   VAR
      b_HmiCmdModAut { ExternalVisible := 'False'} : Bool;   //  command change mode to AUTO
      b_HmiCmdModMan { ExternalVisible := 'False'} : Bool;   //  command change mode to MANUAL
      b_HmiCmdModDis { ExternalVisible := 'False'} : Bool;   //  command change mode to DISABLED
      b_HmiCmdSim { ExternalVisible := 'False'} : Bool;   //  toggle simulation mode
      b_HmiCmdRst { ExternalVisible := 'False'} : Bool;   //  reset alarms
      b_HmiCmdAutoSim { ExternalVisible := 'False'} : Bool;   //  toggle automatic simulation value
      b_HmiCmdFwd { ExternalVisible := 'False'} : Bool;   //  command start forward
      b_HmiCmdRev { ExternalVisible := 'False'} : Bool;   //  command start reversed
      b_HmiCmdStp { ExternalVisible := 'False'} : Bool;   //  command stop
      b_HmiCmdRstActOpe { ExternalVisible := 'False'} : Bool;   //  reset actuation counter and operating hours
      b_StaModAut { ExternalVisible := 'False'} : Bool;   //  state AUTOMATIC
      b_StaModMan { ExternalVisible := 'False'} : Bool := TRUE;   //  state MANUAL
      b_StaModDis { ExternalVisible := 'False'} : Bool;   //  state DISABLED
      b_StaSim { ExternalVisible := 'False'} : Bool;   //  state simulation ON
      b_StaIlOn { ExternalVisible := 'False'} : Bool;   //  state interlock ON : 1 = interlocked (prevents forward)
      b_StaIlRev : Bool;   //  state interlock ON : 1 = interlocked (prevents reverse)
      b_StaSaf { ExternalVisible := 'False'} : Bool;   //  state safety : 1 = error (valve to safety position)
      b_StaAutoSim { ExternalVisible := 'False'} : Bool;   //  Auto sim (Ir_ActSpd simulated)
      b_ReqFwd { ExternalVisible := 'False'} : Bool;   //  output forward
      b_ReqRev { ExternalVisible := 'False'} : Bool;   //  output reversed
      b_StaSpdOk { ExternalVisible := 'False'} : Bool;   //  speed (setpoint) reached
      b_StaAlm { ExternalVisible := 'False'} : Bool;   //  general alarm
      b_StaWrn { ExternalVisible := 'False'} : Bool;   //  general warning
      b_CfgAnaSpdPres { ExternalVisible := 'False'} : Bool;   //  configuration : analog speed feedback present
      b_CfgEnRev { ExternalVisible := 'False'} : Bool;   //  configuration : reversed direction enabled
      b_CfgHldMod { ExternalVisible := 'False'} : Bool;   //  Configuration : status bit mode after reset (1 = auto, 0 = manual)
      b_CfgPushToRun { ExternalVisible := 'False'} : Bool;
      b_CfgDisableSim { ExternalVisible := 'False'} : Bool;
      b_CfgStopArea { ExternalVisible := 'False'} : Bool;
      b_AlmToFb { ExternalVisible := 'False'} : Bool;   //  alarm time out feedback
      b_AlmToRun { ExternalVisible := 'False'} : Bool;   //  alarm run time too long
      b_AlmIs { ExternalVisible := 'False'} : Bool;   //  alarm isolation switch
      b_AlmMps { ExternalVisible := 'False'} : Bool;   //  alarm motor protection switch
      b_AlmDevFlt { ExternalVisible := 'False'} : Bool;   //  alarm device fault
      b_ReqAut { ExternalVisible := 'False'} : Bool;   //  automatic mode requested
      b_ReqMan { ExternalVisible := 'False'} : Bool;   //  manual mode requested
      b_ReqDis { ExternalVisible := 'False'} : Bool;   //  disabled mode requested
      b_TFbSpd { ExternalVisible := 'False'} : Bool;   //  timer finished, feedback monitoring Pos1
      b_SpChange : Bool;
      r_SpSel { ExternalVisible := 'False'} : Real;   //  selected setpoint
      r_SpPrev : Real;
      r_DevMax { ExternalVisible := 'False'} : Real;
      r_DevMin { ExternalVisible := 'False'} : Real;
      b_CmdManFwd { ExternalVisible := 'False'} : Bool;   //  internal memo : manual command forward
      b_CmdManRev { ExternalVisible := 'False'} : Bool;   //  internal memo : manual command reversed
      b_CmdAutFwd { ExternalVisible := 'False'} : Bool;   //  internal memo : automatic command forward
      b_CmdAutRev { ExternalVisible := 'False'} : Bool;   //  internal memo : automatic command reversed
      b_CmdFwd { ExternalVisible := 'False'} : Bool;   //  internal memo : command forward (combined manual and auto)
      b_CmdRev { ExternalVisible := 'False'} : Bool;   //  internal memo : command reversed(combined manual and auto)
      b_FbErrSpd { ExternalVisible := 'False'} : Bool;   //  internal memo : error detection feedback analogue value
      b_TFbOnOut { ExternalVisible := 'False'} : Bool;   //  timer finished for feedback monitoring run (Fwd OR Rev)
      b_TFbOffOut { ExternalVisible := 'False'} : Bool;   //  timer finished for feedback monitoring stop
      b_TToRunOut { ExternalVisible := 'False'} : Bool;   //  timer finished for time out run
      i_TmrToRun : Int;   //  timer time out  run control
      i_TmrFbFwd { ExternalVisible := 'False'} : Int;   //  timer for feedback simulation (set) after start
      i_TmrFbRev { ExternalVisible := 'False'} : Int;   //  timer for feedback simulation (reset) after stop
      b_TFbFwdOut { ExternalVisible := 'False'} : Bool;   //  timer finished for simulation run (Fwd OR Rev)
      b_TFbRevOut { ExternalVisible := 'False'} : Bool;   //  timer finished for simulation stopped
      FB_UTIL_TON_Del_1 : "FB_UTIL_TON_Sec";
      FB_UTIL_TON_Del_2 : "FB_UTIL_TON_Sec";
      FB_UTIL_TON_Del_3 : "FB_UTIL_TON_Sec";
      FB_UTIL_TON_Del_4 : "FB_UTIL_TON_Sec";
      b_Old_ob_Fwd : Bool;
      b_Old_ob_Rev : Bool;
      FB_UTIL_Work_H_Rst { ExternalVisible := 'False'} : "FB_UTIL_Work_H";
      FB_UTIL_Work_H_Tot { ExternalVisible := 'False'} : "FB_UTIL_Work_H";
      b_FbSimFwd : Bool;
      b_FbSimRev : Bool;
      b_FbErrFwd : Bool;
      b_FbErrRev : Bool;
      i_TmrFbSpd : Int;
      b_DisAlmWrn : Bool;
      b_dummy : Bool;
      i_dummy : Int;
      b_StaAlmNew : Bool;
      b_NoAlm : Bool;
      i_AlmAck : Int;
      b_DisAlmWrn_1 : Bool;
      b_RstAlm : Bool;
      b_HmiCmdLoc : Bool;
      b_HmiCmdRem : Bool;
      i_ErrCod : Int;
      b_LocGenEnab : Bool;
      b_DrwTest : Bool;
      b_DrwInst : Bool;
      b_DrwNotIns : Bool;
      b_ErrorCFW : Bool;
      b_RemoteM : Bool;
      b_ManutLocal { ExternalVisible := 'False'} : Bool;   // command change mode to "Manut.Local"
      b_FbRem : Bool;
      b_PerRemMod : Bool;
      I_HmiSta : Word;
      i_Category : Int := 1;   // Device alarm category setting
      b_NoFeedback : Bool;
      b_EnDisPump : Bool;   // Enable/Disable HMI option
   END_VAR

   VAR_TEMP
      di_AUX : DInt;   //  auxiliary double word for calculation of state or alarm word to HMI
   END_VAR


BEGIN
	// =============================================================================================================================
	// Purpose: Reditech standard typical for controlling a frequency driven motor
	// -----------------------------------------------------------------------------------------------------------------------------
	// Date (dd MMM yyyy)   Developer                   Version Comments/Reason for change
	// ..................   .........                   ....... ..........................
	// 13 Dec 2018          Bram Verheyen               08.0    Full review
	// 30 Jan 2019          Matthias De Staelen         08.1    Outputs can be high in simulation mode
	// 13 Mar 2020          Willian Barroso             08.2    Full review
	// 01 Jul 2021          Ivan Galhardoni             08.3    Added NoFeedback function
	// 03 Jul 2021          Ivan Galhardoni             08.4    Added No communication fault alarm and erase manual setpoint when interlock is incoming
	// =============================================================================================================================

	//============================================================================================
	#b_CfgAnaSpdPres := #Iw_Cfg.%X0;      // Analog speed feedback present
	#b_CfgEnRev := #Iw_Cfg.%X1;           // Reverse direction enable
	#b_CfgHldMod := #Iw_Cfg.%X2;          // Mode after reset (1 => auto, 0 => manual)
	#b_NoFeedback := #Iw_Cfg.%X3;         // No feedback configured
	#b_CfgPushToRun := #Iw_Cfg.%X8;
	#b_CfgDisableSim := #Iw_Cfg.%X10;
	#b_CfgStopArea := #Iw_Cfg.%X11;

	//============================================================================================
	#b_DisAlmWrn := #Ib_DisAlmWrn OR #IO_AreaCmd.Alm.Dis OR #b_StaModDis OR #b_StaSim;

	//============================================================================================
	#b_StaSaf := (#Iby_Saf <> 0) AND NOT #b_DisAlmWrn;
	#b_StaIlOn := (#Iby_IlFwd <> 0);
	//#b_StaIlRev := (#Iby_IlRev <> 0);

	//============================================================================================
	IF #b_StaSim THEN
	    #i_ErrCod := 15;
	    #b_LocGenEnab := TRUE;
	    #b_FbRem := TRUE;
	ELSE
	    #i_ErrCod := #Ii_CurFault;
	    #b_LocGenEnab := #Ib_LocGenEnab;
	    #b_FbRem := #Ib_FbRem;
	END_IF;

	#b_DrwTest := #Ib_DrwTest;
	#b_DrwInst := #Ib_DrwInst;

	//============================================================================================
	#b_HmiCmdModAut := #IOdi_HmiCmd.%X0;
	#b_HmiCmdModMan := #IOdi_HmiCmd.%X1;
	#b_HmiCmdModDis := #IOdi_HmiCmd.%X2;
	#b_HmiCmdSim := #IOdi_HmiCmd.%X3;
	#b_HmiCmdFwd := #IOdi_HmiCmd.%X4;
	#b_HmiCmdRev := #IOdi_HmiCmd.%X5;
	#b_HmiCmdStp := #IOdi_HmiCmd.%X6;
	#b_HmiCmdAutoSim := #IOdi_HmiCmd.%X8;
	#b_HmiCmdRstActOpe := #IOdi_HmiCmd.%X9;
	#b_ManutLocal := #IOdi_HmiCmd.%X10;

	//============================================================================================

	IF #b_CfgPushToRun THEN
	    #IOdi_HmiCmd := DWORD_TO_DINT(DINT_TO_DWORD(#IOdi_HmiCmd) AND 48);
	ELSE
	    #IOdi_HmiCmd := 0;
	END_IF;


	//============================================================================================
	IF  #IO_AreaCmd.Mode.AreaMode THEN
	    #b_ReqAut := #IO_AreaCmd.Mode.Auto;
	    #b_ReqMan := #IO_AreaCmd.Mode.Man;
	    #b_ReqDis := #IO_AreaCmd.Mode.Dis;

	ELSE
	    IF #b_CfgHldMod THEN
	        #b_ReqAut := #b_HmiCmdModAut;
	        #b_ReqMan := #b_HmiCmdModMan;
	        #b_ReqDis := #b_HmiCmdModDis;

	    ELSE
	        #b_ReqAut := #b_HmiCmdModAut AND NOT #b_StaAlm AND NOT #b_StaSaf;
	        #b_ReqMan := #b_HmiCmdModMan OR ((#b_StaAlm OR #b_StaSaf) AND NOT #b_StaModDis);
	        #b_ReqDis := #b_HmiCmdModDis;
	    END_IF;
	END_IF;
	IF (#b_ReqAut AND NOT #b_ReqMan AND NOT #b_ReqDis) THEN
	    #b_StaModAut := true;
	    #b_StaModMan := false;
	    #b_StaModDis := false;
	END_IF;
	IF (#b_ReqMan AND NOT #b_ReqAut AND NOT #b_ReqDis) THEN
	    #b_StaModAut := false;
	    #b_StaModMan := true;
	    #b_StaModDis := false;
	END_IF;
	IF (#b_ReqDis AND NOT #b_ReqMan AND NOT #b_ReqAut) THEN
	    #b_StaModAut := false;
	    #b_StaModMan := false;
	    #b_StaModDis := true;
	END_IF;

	//============================================================================================
	IF #IO_AreaCmd.Sim.ForceOn OR (#b_HmiCmdSim AND NOT #b_StaSim AND NOT #IO_AreaCmd.Sim.ForceOn AND NOT #IO_AreaCmd.Sim.ForceOff) THEN
	    #b_StaSim := true;
	    #b_HmiCmdSim := false; // reset of command necessary, else simulation will always be reset immediately by following instructions
	END_IF;
	IF #IO_AreaCmd.Sim.ForceOff OR (#b_HmiCmdSim AND #b_StaSim AND NOT #IO_AreaCmd.Sim.ForceOn AND NOT #IO_AreaCmd.Sim.ForceOff) THEN
	    #b_StaSim := false;
	    #b_HmiCmdSim := false;
	END_IF;

	//============================================================================================
	IF (#b_ReqFwd AND NOT #b_FbSimFwd)
	    OR (#b_ReqRev AND NOT #b_FbSimRev)
	    OR #b_HmiCmdStp
	    OR (NOT #b_ReqFwd AND NOT #b_ReqRev)
	    OR #b_StaIlOn
	    OR #b_StaAlm THEN
	    #b_FbSimFwd := false;
	    #b_FbSimRev := false;
	END_IF;

	IF ((#i_TmrFbFwd <= 1) OR #Ii_ParTFb = 0) AND #b_ReqFwd THEN
	    #b_FbSimFwd := true;
	    #b_FbSimRev := false;
	END_IF;

	IF ((#i_TmrFbRev <= 1) OR #Ii_ParTFb = 0) AND #b_ReqRev THEN
	    #b_FbSimFwd := false;
	    #b_FbSimRev := true;
	END_IF;

	//============================================================================================
	#r_DevMax := #r_SpSel + #Ir_ParCtlDev;
	#r_DevMin := #r_SpSel - #Ir_ParCtlDev;
	IF #b_StaSim AND #Ib_Pls1S THEN
	    IF (#IOr_SimSpd <= #r_DevMin) THEN
	        #IOr_SimSpd := #IOr_SimSpd + #Ir_ParCtlDev;
	    END_IF;
	    IF (#IOr_SimSpd >= #r_DevMax) THEN
	        #IOr_SimSpd := #IOr_SimSpd - #Ir_ParCtlDev;
	    END_IF;
	END_IF;

	// ACM: select speed
	IF #b_StaSim THEN
	    #Or_StaSpd := #IOr_SimSpd;
	ELSE
	    #Or_StaSpd := #Ir_ActSpd;
	END_IF;

	//============================================================================================
	#Ob_StaFwd := (NOT #b_StaSim AND #Ib_FbFwd)
	OR (#b_StaSim AND #b_FbSimFwd)
	OR (#b_NoFeedback AND #r_SpSel > 0.00);

	#Ob_StaRev := (NOT #b_StaSim AND #Ib_FbRev)
	OR (#b_StaSim AND #b_FbSimRev);

	#Ob_StaOff := NOT #Ob_StaFwd AND NOT #Ob_StaRev;

	#b_StaSpdOk := (NOT #b_CfgAnaSpdPres)
	OR (#b_CfgAnaSpdPres AND (#Or_StaSpd > #r_DevMin) AND (#Or_StaSpd < #r_DevMax));
	#Ob_SpdOk := #b_StaSpdOk AND NOT #b_StaAlm;

	//============================================================================================
	#b_SpChange := (#r_SpSel <> #r_SpPrev);
	#r_SpPrev := #r_SpSel;

	//============================================================================================
	#b_NoAlm := false;
	#b_RstAlm := #b_HmiCmdRst OR #IO_AreaCmd.Alm.Rst;
	"FC_UTIL_AlmAck"(Ib_CmdAck := #b_RstAlm,
	                 Oi_StaAlm => #i_dummy,
	                 Ob_StaAlm => #b_dummy,
	                 Ob_StaNewAlm => #b_StaAlmNew,
	                 IO_Alm0 := #b_AlmToFb,
	                 IO_Alm1 := #b_AlmToRun,
	                 IO_Alm2 := #b_AlmIs,
	                 IO_Alm3 := #b_AlmMps,
	                 IO_Alm4 := #b_StaWrn,
	                 IO_Alm5 := #b_AlmDevFlt,
	                 IO_Alm6 := #b_ErrorCFW,
	                 IO_Alm7 := #b_DrwNotIns,
	                 IO_Alm8 := #b_NoAlm,
	                 IO_Alm9 := #b_NoAlm,
	                 IO_Alm10 := #b_NoAlm,
	                 IO_Alm11 := #b_NoAlm,
	                 IO_Alm12 := #b_NoAlm,
	                 IO_Alm13 := #b_NoAlm,
	                 IO_Alm14 := #b_NoAlm,
	                 IO_Alm15 := #b_NoAlm,
	                 IOi_StaAck := #i_AlmAck);

	//============================================================================================
	IF (#Ii_ParTFb > 0) THEN  // only when time value > 0
	    #FB_UTIL_TON_Del_1(Ii_tValue := #Ii_ParTFb,
	                       Ib_In := (#b_ReqFwd AND NOT #Ob_StaFwd),
	                       Ii_Base := 1,
	                       Ib_Hold := 0,
	                       Ob_Out => #b_FbErrFwd,
	                       Oi_tmrValue => #i_TmrFbFwd);
	END_IF;

	IF (#Ii_ParTFb > 0) THEN  // only when time value > 0
	    #FB_UTIL_TON_Del_2(Ii_tValue := #Ii_ParTFb,
	                       Ib_In := (#b_ReqRev AND NOT #Ob_StaRev),
	                       Ii_Base := 1,
	                       Ib_Hold := 0,
	                       Ob_Out => #b_FbErrRev,
	                       Oi_tmrValue => #i_TmrFbRev);
	END_IF;

	IF (#Ii_ParTO > 0) THEN
	    #FB_UTIL_TON_Del_4(Ib_In := (#b_CfgAnaSpdPres AND NOT #b_StaSpdOk AND NOT #b_SpChange AND (#b_ReqFwd OR #b_ReqRev)),
	                       Ii_tValue := #Ii_ParTO,
	                       Ii_Base := 1,
	                       Ib_Hold := 0,
	                       Ob_Out => #b_FbErrSpd,
	                       Oi_tmrValue => #i_TmrFbSpd);
	END_IF;

	IF (((#b_FbErrFwd OR #b_FbErrRev) AND (#Ii_ParTFb > 0))
	    OR (#b_FbErrSpd AND (#Ii_ParTO > 0)))
	    AND NOT #b_DisAlmWrn THEN
	    #b_AlmToFb := true;
	END_IF;

	//============================================================================================
	IF (#Ii_ParTToRun > 0) THEN
	    #FB_UTIL_TON_Del_3(Ii_tValue := #Ii_ParTToRun,
	                       Ib_In := (#b_ReqFwd OR #b_ReqRev),
	                       Ii_Base := 1,
	                       Ib_Hold := 0,
	                       Ob_Out => #b_TToRunOut,
	                       Oi_tmrValue => #i_TmrToRun);
	END_IF;

	IF (#b_TToRunOut AND (#Ii_ParTToRun > 0))
	    AND NOT #b_DisAlmWrn THEN
	    #b_AlmToRun := true;
	END_IF;

	//============================================================================================
	IF #ib_Is AND NOT #b_DisAlmWrn THEN
	    #b_AlmIs := true;
	END_IF;

	//============================================================================================
	IF #Ib_Mps AND NOT #b_DisAlmWrn THEN
	    #b_AlmMps := true;
	END_IF;

	//============================================================================================
	IF #Ib_DevFlt AND NOT #b_DisAlmWrn THEN
	    #b_AlmDevFlt := true;
	END_IF;

	//============================================================================================
	IF NOT #b_DrwInst AND NOT #b_DrwTest AND NOT #b_DisAlmWrn THEN
	    #b_DrwNotIns := true;
	END_IF;

	//============================================================================================
	IF (#i_ErrCod = 10) OR (#i_ErrCod = 46) OR (#i_ErrCod = 47) OR (#i_ErrCod = 50) OR
	    (#i_ErrCod = 53) OR (#i_ErrCod = 56) OR (#i_ErrCod = 78) OR (#i_ErrCod = 80) OR (#i_ErrCod = 84) OR
	    (#i_ErrCod = 88) OR (#i_ErrCod = 99) OR (#i_ErrCod = 110) OR (#i_ErrCod = 129) OR
	    (#i_ErrCod = 130) OR (#i_ErrCod = 151) OR (#i_ErrCod = 152) OR (#i_ErrCod = 160) OR
	    (#i_ErrCod = 177) OR (#i_ErrCod = 179) OR (#i_ErrCod = 182) OR (#i_ErrCod = 700) OR
	    (#i_ErrCod = 701) AND NOT #b_DisAlmWrn
	THEN
	    #b_ErrorCFW := true;
	END_IF;

	//============================================================================================
	#b_StaAlm := #b_AlmToFb OR #b_AlmToRun OR #b_StaSaf OR #b_AlmIs OR #b_AlmMps OR #b_DrwNotIns
	OR #b_ErrorCFW OR #b_AlmDevFlt OR NOT #b_EnDisPump;
	#Ob_Alm := #b_StaAlm;

	//============================================================================================
	#b_StaWrn := (#r_SpSel < #Ir_ParMinSpd) OR (#r_SpSel > #Ir_ParMaxSpd);
	#Ob_Wrn := #b_StaWrn;

	//============================================================================================
	#b_CmdAutFwd := (#Ib_AutFwd AND NOT #Ib_AutRev AND NOT #Ob_Rev);
	#b_CmdAutRev := (#Ib_AutRev AND NOT #Ib_AutFwd AND NOT #Ob_Fwd) AND #b_CfgEnRev;


	IF #b_StaModAut THEN
	    #b_CmdManFwd := #b_CmdAutFwd;
	    #b_CmdManRev := #b_CmdAutRev;
	END_IF;

	//============================================================================================
	IF #b_StaModMan AND NOT #b_CfgPushToRun THEN
	    IF (#b_HmiCmdFwd AND NOT #Ob_Rev) THEN
	        #b_CmdManFwd := true;
	        #b_CmdManRev := false;
	    END_IF;
	    IF (#b_HmiCmdRev AND NOT #Ob_Fwd AND #b_CfgEnRev) THEN
	        #b_CmdManFwd := false;
	        #b_CmdManRev := true;
	    END_IF;
	    IF #b_HmiCmdStp OR #b_StaAlm OR #b_StaModDis OR #b_StaIlOn THEN
	        #b_CmdManFwd := false;
	        #b_CmdManRev := false;
	    END_IF;
	END_IF;

	IF #b_StaModMan AND #b_CfgPushToRun THEN
	    #b_CmdManFwd := #b_HmiCmdFwd AND NOT #Ob_Rev AND NOT #b_StaAlm AND NOT #b_StaModDis;
	    #b_CmdManRev := #b_HmiCmdRev AND NOT #Ob_Fwd AND NOT #b_StaAlm AND NOT #b_StaModDis AND #b_CfgEnRev;
	END_IF;

	IF #b_StaModDis OR NOT #b_StaModMan THEN
	    #b_CmdManFwd := false;
	    #b_CmdManRev := false;
	END_IF;

	//============================================================================================
	IF #b_StaModAut THEN
	    #r_SpSel := #IOr_AutSp;
	    #IOr_ManSP := #IOr_AutSp;
	END_IF;

	IF #b_StaModMan THEN
	    #r_SpSel := #IOr_ManSP;
	END_IF;

	IF #b_StaModDis OR #b_StaAlm OR #b_StaIlOn THEN
	    #r_SpSel := 0.0;
	    #IOr_ManSP := 0.0;
	END_IF;

	IF #b_StaSaf THEN
	    #r_SpSel := #Ir_ParSafSpd;
	END_IF;

	#r_SpSel := LIMIT(MN := #Ir_ParMinSpd, IN := #r_SpSel, MX := #Ir_ParMaxSpd);

	//============================================================================================
	#b_CmdFwd := (#b_StaModAut AND #b_CmdAutFwd) OR (#b_StaModMan AND #b_CmdManFwd) OR (#b_NoFeedback AND #r_SpSel > 0.00);
	#b_CmdRev := (#b_StaModAut AND #b_CmdAutRev) OR (#b_StaModMan AND #b_CmdManRev);

	//============================================================================================
	#b_ReqFwd := (#b_CmdFwd AND NOT #b_StaAlm AND NOT #b_StaIlOn AND NOT #b_StaModDis);
	#b_ReqRev := (#b_CmdRev AND NOT #b_StaAlm AND NOT #b_StaIlOn AND NOT #b_StaModDis);

	//============================================================================================
	IF #b_StaSim THEN
	    #Ob_Fwd := FALSE;
	    #Ob_Rev := FALSE;
	ELSE
	    #Ob_Fwd := #b_ReqFwd;
	    #Ob_Rev := #b_ReqRev;
	END_IF;
	#Ob_Off := NOT #b_ReqFwd AND NOT #b_ReqRev;

	IF #Ob_StaFwd THEN
	    #Or_SpOut := #r_SpSel;
	ELSE
	    #Or_SpOut := 0.0;
	END_IF;


	//============================================================================================
	#Odi_HmiSta.%X0 := #b_StaModAut;
	#Odi_HmiSta.%X1 := #b_StaModMan;
	#Odi_HmiSta.%X2 := #b_StaModDis;
	#Odi_HmiSta.%X3 := #b_StaSim;
	#Odi_HmiSta.%X4 := #b_StaIlOn OR #b_StaSaf;
	#Odi_HmiSta.%X5 := #b_StaIlRev;
	#Odi_HmiSta.%X6 := #b_StaSaf AND NOT #b_AlmDevFlt;
	#Odi_HmiSta.%X7 := #b_StaAutoSim;
	#Odi_HmiSta.%X8 := #b_LocGenEnab;
	#Odi_HmiSta.%X9 := #b_DrwTest;
	#Odi_HmiSta.%X12 := #b_FbRem;
	#Odi_HmiSta.%X15 := #b_StaSpdOk;
	#Odi_HmiSta.%X16 := #b_ReqFwd;
	#Odi_HmiSta.%X17 := #b_ReqRev;
	#Odi_HmiSta.%X18 := #Ob_StaFwd;
	#Odi_HmiSta.%X19 := #Ob_StaRev;
	#Odi_HmiSta.%X20 := #b_StaAlm;
	#Odi_HmiSta.%X21 := #b_StaWrn;
	#Odi_HmiSta.%X28 := #IO_AreaCmd.Mode.AreaMode;
	#Odi_HmiSta.%X29 := #b_PerRemMod;

	#I_HmiSta.%X0 := #b_StaModAut;
	#I_HmiSta.%X1 := #b_StaModMan;
	#I_HmiSta.%X2 := #b_StaModDis;
	#I_HmiSta.%X3 := #b_StaSim;
	#I_HmiSta.%X4 := #b_StaIlOn OR #b_StaSaf;
	#I_HmiSta.%X5 := #b_StaSaf;
	#I_HmiSta.%X6 := #b_LocGenEnab;
	#I_HmiSta.%X7 := #b_FbRem;
	#I_HmiSta.%X8 := #Ob_StaFwd;
	#I_HmiSta.%X9 := #b_StaAlm;

	//============================================================================================
	#di_AUX := 0;
	#di_AUX.%X0 := #b_AlmToFb;
	#di_AUX.%X1 := #b_AlmToRun;
	#di_AUX.%X2 := #b_AlmIs AND NOT #b_AlmDevFlt;
	#di_AUX.%X3 := #b_AlmMps AND NOT #b_AlmDevFlt;
	#di_AUX.%X4 := #b_StaWrn;
	#di_AUX.%X5 := #b_AlmDevFlt;
	#di_AUX.%X6 := #b_DrwNotIns AND NOT #b_AlmDevFlt;
	#di_AUX.%X7 := #b_ErrorCFW AND NOT #b_AlmDevFlt;
	#di_AUX.%X16 := #Iby_IlFwd.%X0;
	#di_AUX.%X17 := #Iby_IlFwd.%X1;
	#di_AUX.%X18 := #Iby_IlFwd.%X2;
	#di_AUX.%X19 := #Iby_IlFwd.%X3;
	#di_AUX.%X20 := #Iby_IlFwd.%X4;
	#di_AUX.%X21 := #Iby_IlFwd.%X5;
	#di_AUX.%X22 := #Iby_IlFwd.%X6;
	#di_AUX.%X23 := #Iby_IlFwd.%X7;
	#di_AUX.%X24 := #Iby_Saf.%X0;
	#di_AUX.%X25 := #Iby_Saf.%X1;
	#di_AUX.%X26 := #Iby_Saf.%X2;
	#di_AUX.%X27 := #Iby_Saf.%X3;
	#di_AUX.%X28 := #Iby_Saf.%X4;
	#di_AUX.%X29 := #Iby_Saf.%X5;
	#di_AUX.%X30 := #Iby_Saf.%X6;
	#di_AUX.%X31 := #Iby_Saf.%X7;
	#Odi_HmiAlm := #di_AUX;

	//============================================================================================
	#di_AUX := 0;
	#di_AUX.%X0 := #b_AlmToFb;
	#di_AUX.%X1 := #b_AlmToRun AND NOT #b_AlmDevFlt;
	#di_AUX.%X2 := #b_AlmIs AND NOT #b_AlmDevFlt;
	#di_AUX.%X3 := #b_AlmMps AND NOT #b_AlmDevFlt;
	#di_AUX.%X4 := #b_StaWrn;
	#di_AUX.%X5 := #b_AlmDevFlt;
	#Oi_HmiAlm := DINT_TO_INT(#di_AUX);

	//============================================================================================
	IF #b_StaModDis THEN
	    #IO_AreaFb.Mode.Dis := TRUE;
	END_IF;
	IF #b_StaModMan THEN
	    #IO_AreaFb.Mode.Man := TRUE;
	END_IF;
	IF #b_StaModAut THEN
	    #IO_AreaFb.Mode.Auto := TRUE;
	END_IF;
	IF #b_StaAlm THEN
	    #IO_AreaFb.Alm.Alm := TRUE;
	END_IF;
	IF #b_StaAlmNew THEN
	    #IO_AreaFb.Alm.New := TRUE;
	END_IF;
	IF #b_StaWrn THEN
	    #IO_AreaFb.Alm.Wrn := TRUE;
	END_IF;
	IF #b_StaAlm AND #b_CfgStopArea THEN
	    #IO_AreaFb.Alm.StopArea := TRUE;
	END_IF;

	//Generating alarm category feedback
	IF #i_Category = 1 AND #b_StaAlm THEN
	    #IO_AreaFb.Alm.Alm_Lvl1 := TRUE;
	END_IF;

	IF #i_Category = 2 AND #b_StaAlm THEN
	    #IO_AreaFb.Alm.Alm_Lvl2 := TRUE;
	END_IF;

	IF #i_Category = 3 AND #b_StaAlm THEN
	    #IO_AreaFb.Alm.Alm_Lvl3 := TRUE;
	END_IF;

	//============================================================================================
	IF (#Ob_Fwd <> #b_Old_ob_Fwd) OR (#Ob_Rev <> #b_Old_ob_Rev) THEN
	    #Odi_ActCouRst := #Odi_ActCouRst + 1;
	    #Odi_ActCouTot := #Odi_ActCouTot + 1;
	END_IF;
	IF #b_HmiCmdRstActOpe THEN
	    #Odi_ActCouRst := 0;
	END_IF;
	#b_Old_ob_Fwd := #Ob_Fwd;
	#b_Old_ob_Rev := #Ob_Rev;

	//============================================================================================
	//Local/Remote Operation
	IF #b_RemoteM AND #b_ManutLocal THEN
	    #b_RemoteM := FALSE;
	ELSIF NOT #b_RemoteM AND #b_ManutLocal THEN
	    #b_RemoteM := TRUE;
	END_IF;

	#Ob_LocRem := #b_RemoteM;

	//Local/Remote Operation
	IF #b_StaModMan AND NOT #b_StaModAut AND NOT #b_StaModDis THEN
	    #b_PerRemMod := TRUE;
	ELSE
	    #b_PerRemMod := FALSE;
	END_IF;

	//============================================================================================
	#FB_UTIL_Work_H_Rst(Ib_On := #Ob_Fwd OR #Ob_Rev,
	                    Ib_Reset := #b_HmiCmdRstActOpe,
	                    Ib_Pls1S := "Clock_1Hz",
	                    IOdi_ResultHours := #Odi_RunTimRst);

	#FB_UTIL_Work_H_Tot(Ib_On := #Ob_Fwd OR #Ob_Rev,
	                    Ib_Pls1S := "Clock_1Hz",
	                    IOdi_ResultHours := #Odi_RunTimTot);
END_FUNCTION_BLOCK

FUNCTION_BLOCK "G120C_Tel20"
{ S7_Optimized_Access := 'TRUE' }
VERSION : 0.1
   VAR_INPUT DB_SPECIFIC
      EM_Stop : Bool;   // 0 - parada de emergência ativa
      Release : Bool;   // Liberação do motor para operar
      Mode : Bool;   // 1 - Auto /0 - Manual
      Start_FW : Bool;   // Comando para avançar em automático
      Start_RV : Bool;   // Comando para recuar em automático
      Start_Man_FW : Bool;   // Comando para avançar em manual
      Start_MAN_RV : Bool;   // Comando para recuar em manual
      Reset : Bool;   // Reset de falhas do inversor
      SP : Real;   // Setpoint de velocidade do inversor em %
      SP_Man : Real;   // Setpoint de velocidade em modo manual do inversor em %
      G120_ZSW : Word;   // Status word do G120
      G120_NIST_A : Int;   // Velocidade atual do G120
      G120_IAIST : Int;   // Corrente atual do G120
      G120_MIST : Int;   // Torque atual do G120
      G120_F_Ref : Real;   // Referência do sinal de frequência
      G120_I_Ref : Real;   // Referência do sinal de corrente
      G120_T_Ref : Real;   // Referência do sinal de torque
   END_VAR

   VAR_OUTPUT DB_SPECIFIC
      Rdy_Start : Bool;   // Inversor ligado e inicializado
      Rdy : Bool;   // Inversor pronto para operar
      Enabled : Bool;   // Inversor seguindo o SP
      Fault : Bool;   // Inversor em falha
      OFF2 : Bool;   // Parada por inercia não ativa
      OFF3 : Bool;   // Parada rápida não ativa
      Alarm : Bool;   // Inversor em alarme
      SP_OK : Bool;   // Inversor está no SP
      Dir : Bool;   // 1 - Direto / 0 - Reverso
      EM_Fault : Bool;
      G120_STW : Word;   // Palavra de comando do inversor
      G120_NSOLL_A : Int;   // SP do inversor
      Freq : Real;   // Frequência atual do motor
      Curr : Real;   // Corrente atual do motor
      Torq : Real;   // Torque atual do motor
   END_VAR

   VAR_IN_OUT DB_SPECIFIC
      Lockout : Bool;
      Mater_Ctrl_Req : Bool;
      Max_Speed : Bool;
      FW_OK : Bool;
      RV_OK : Bool;
   END_VAR

   VAR_TEMP
      Aux_Conv : Word;   // Auxiliar para converter word para bit e vice versa
      Aux_Int : Int;
      G120_STW_Aux : Word;   // Auxiliar para montar palavra de comando do inversor
      Aux_Conv_DI : DInt;   // Auxiliar para convertar 0 - 16X4000 para 0-100 e vice versa
      Aux_Conv_R : Real;   // Auxiliar para convertar 0 - 16X4000 para 0-100 e vice versa
      Temp : Int;
   END_VAR


BEGIN
	// =============================================================================================================================
	// Purpose: G120C inverter telegram 20 communication block
	// -----------------------------------------------------------------------------------------------------------------------------
	// Date (dd MMM yyyy)   Developer                   Version   Comments/Reason for change
	// ..................   .........                   ....... ..........................
	// 22 Jan 2025          Gustavo Lourenção             01      Block language switch (Ladder to SCL)
	//
	// -----------------------------------------------------------------------------------------------------------------------------
	// =============================================================================================================================
	//
	// ------------------------- ATENÇÃO* BLOCO COM O FUNCIONAMENTO AINDA NÃO VALIDADO, SE NÃO FUNCIONAR COPIE O G120C_TEL20 COM A LINGUAGEM LADDER---------------------

	#G120_STW_Aux := Int#0 ; //
	#G120_STW := #G120_STW_Aux; // copia palavra de comando

	// Detecta parada de emergencia e reseta a falha
	IF #EM_Stop THEN
	    // Statement section IF
	    #EM_Fault := 1;
	ELSIF #Reset THEN
	    #EM_Fault := 0;
	END_IF;


	#Rdy_Start := #G120_ZSW.%X0;
	#Rdy := #G120_ZSW.%X1;
	#Enabled := #G120_ZSW.%X2;
	#Fault := #G120_ZSW.%X3;
	#OFF2 := #G120_ZSW.%X4;
	#OFF3 := #G120_ZSW.%X5;
	#Lockout := #G120_ZSW.%X6;
	#Alarm := #G120_ZSW.%X7;
	#SP_OK := #G120_ZSW.%X8;
	#Mater_Ctrl_Req := #G120_ZSW.%X9;
	#Max_Speed := #G120_ZSW.%X10;
	#Dir := #G120_ZSW.%X14;


	#G120_STW_Aux.%X0 := #FW_OK OR #RV_OK; //OFF1 Ctr
	#G120_STW_Aux.%X1 := TRUE; //OFF 2 sempre ativo
	#G120_STW_Aux.%X2 := NOT #EM_Fault; //OFF3 (em caso de parada de emergência)
	#G120_STW_Aux.%X3 := #Release; //Enable (Release de operação)
	#G120_STW_Aux.%X4 :=
	#G120_STW_Aux.%X5 := TRUE; //Do not disable RFG/Enable RFG/ Enable SP/Control  (sempre ativo)
	#G120_STW_Aux.%X6 := TRUE; //Do not disable RFG/Enable RFG/ Enable SP/Control  (sempre ativo)
	#G120_STW_Aux.%X7 := #Reset;
	#G120_STW_Aux.%X8 :=
	#G120_STW_Aux.%X9 :=
	#G120_STW_Aux.%X10 :=
	#G120_STW_Aux.%X11 := #RV_OK AND NOT #FW_OK;
	#G120_STW_Aux.%X12 :=
	#G120_STW_Aux.%X13 :=
	#G120_STW_Aux.%X14 := TRUE; //Do not disable RFG/Enable RFG/ Enable SP/Control  (sempre ativo)
	#G120_STW_Aux.%X15 := FALSE;

	//Calcula SP auto para o inversor
	IF #Mode AND #SP >= 115.0 THEN
	    #G120_NSOLL_A := W#16#4000;
	END_IF;

	IF #Mode AND #SP <= 0 THEN
	    #G120_NSOLL_A := 0;
	END_IF;

	IF #Mode AND #SP > 0 AND #SP <= 115.0 THEN
	    #Aux_Conv_R := #SP * 163.84;
	END_IF;

	//Calcula #SP manual para inversor
	IF NOT #Mode AND #SP_Man >= 100.0 THEN
	    #Aux_Conv_R := 100.0;
	END_IF;

	IF NOT #Mode AND #SP_Man <= 0.0 THEN
	    #Aux_Conv_R := 0.0;
	END_IF;

	IF NOT #Mode AND #SP_Man > 0 AND #SP_Man <= 100.0 THEN
	    #Aux_Conv_R := #SP_Man * 163.84;
	END_IF;

	//converte SP e envia para drive
	#Aux_Conv_DI := ROUND(#Aux_Conv_R);
	#G120_NSOLL_A := #Aux_Conv_DI;

	//Converte sinal de Corrente
	#Aux_Conv_DI := INT_TO_DINT(#G120_NIST_A);
	#Aux_Conv_R := DINT_TO_REAL(#Aux_Conv_DI) / 16384.0;
	#Freq := #Aux_Conv_R * #G120_F_Ref;

	#Aux_Conv_DI := INT_TO_DINT(#G120_IAIST);
	#Aux_Conv_R := DINT_TO_REAL(#Aux_Conv_DI) / 16384.0;
	#Curr := #Aux_Conv_R * #G120_I_Ref;

	#Aux_Conv_DI := INT_TO_DINT(#G120_MIST);
	#Aux_Conv_R := DINT_TO_REAL(#Aux_Conv_DI) / 16384.0;
	#Torq := #Aux_Conv_R * #G120_T_Ref;

	//Start Fw
	#FW_OK := (#Mode AND #Start_FW) OR (NOT #Mode AND #Start_Man_FW) AND #Rdy_Start AND #OFF2 AND #OFF3 AND #Release AND #EM_Stop AND NOT #RV_OK AND NOT #Fault;

	//Start RV
	#RV_OK := (#Mode AND #Start_RV) OR (NOT #Mode AND #Start_MAN_RV) AND #Rdy_Start AND #OFF2 AND #OFF3 AND #Release AND #EM_Stop AND NOT #FW_OK AND NOT #Fault;

END_FUNCTION_BLOCK
